# EPICS substitutions: evrSupport/Db/ioc/bsaGENEdef2.substitutions
#==============================================================================
#
# Abs:  Beam Synchronous Acquisition records for a single
#	    RF Amplitude measurement.
#
# Name: bsaAMPLEdef.substitutions
#
# Note: Must follow the LCLS naming conventions.
#
#==============================================================================
#
#
file bsaATTREdef2.db
{
#           Device   Attribute  Input  EGU   HOPR  LOPR PREC ADEL  Link
  pattern {   D       , ATTR   , I   , EG ,  HO  , LO , PR , AD  ,  LNK             }
	  { $(DEVICE) ,$(ATRB) ,$(IN), $(EGU) , $(HOPR), $(LOPR), $(PREC), $(ADEL)  }
}
